{attribute 'qualified_only'}
{attribute 'strict'}
{attribute 'to_string'}
// TODO - adapt to PackML (?)
TYPE EOperatingModes :
(
	none := 0,
	init := 1,
	automatic := 2,
	manual := 3,
	recovering := 4,
	shutting_down := 5,
	shutdown := 6,
	custom_sequence := 7
) UINT;
END_TYPE

(* stored: Version 1.1.0.1, ProductVersion 3.1.4024.12
   DUT EOperatingModes: Id {ac1d99ed-5793-4b33-b5a6-3d039dcffed1} *)
